// TwinCAT 3 PLC project Untitled1
// ProgramVersion: 3.1.4018.58
// libraries:
//   Tc2_Standard, * (Beckhoff Automation GmbH)
//   Tc2_System, * (Beckhoff Automation GmbH)
//   Tc2_Utilities, * (Beckhoff Automation GmbH)
//   Tc3_Module, * (Beckhoff Automation GmbH)
// project tree:
//   / PlcTask.TcTTO
//   POUs/ FB_GetEndTime.TcPOU, F_GetRampUpTimeString.TcPOU, FB_GetTimeString.TcPOU, MAIN.TcPOU
// real-time tasks:
//   TASK PlcTask: cycle T#10ms, priority 20, ADS port 350

CONFIGURATION Untitled1
    RESOURCE PLC ON TwinCAT3
        TASK PlcTask(INTERVAL := T#10ms, PRIORITY := 20);
        PROGRAM MAIN WITH PlcTask : MAIN;
    END_RESOURCE
END_CONFIGURATION

// ---- POUs/MAIN.TcPOU
PROGRAM MAIN
VAR
	bBool	: BOOL;
	iInt	: INT;
	
	fbGetEndTime: FB_GetEndTime;
	
	bTestTimeCalc	: BOOL;
	strEndTimeString	: STRING(255);
	strStartTimeString	: STRING(255);
	
	bTestGetTimeString	: BOOL;
	strTimeString		: STRING(255);
	fHours				: LREAL	:= 1.26;
END_VAR

iInt	:= iInt + 1;
IF(iInt > 100) THEN
	bBool	:= NOT(bBool); 
	iInt	:= 0;
END_IF

fbGetEndTime();
IF(bTestTimeCalc)THEN
	strEndTimeString	:= fbGetEndTime.GetEndTimeString(3900);
	bTestTimeCalc	:= FALSE;
END_IF

IF(bTestGetTimeString) THEN
	strTimeString		:= fbGetEndTime.GetTimeString(fHours);
	bTestGetTimeString	:= FALSE;
END_IF

END_PROGRAM

// ---- POUs/FB_GetEndTime.TcPOU
FUNCTION_BLOCK FB_GetEndTime	
VAR_INPUT
END_VAR
VAR
	
	// Variables for get end time
	
	diMinutesToWait		: DINT;
	ftTargetTime		: T_FILETIME64;
	stTargetTime		: TIMESTRUCT;
	strTargetTimeString		: STRING(255);
	strPrettyEndTimeString	: STRING(255);
	
	strYear	: STRING;
	strMonth: STRING;
	strDay	: STRING;
	strHour	: STRING;
	strMinute: STRING;
	strSecond: STRING;
	strMiliSecond: STRING;
	
	
	taYear	: T_Arg;
	taMonth : T_Arg;
	taDay	: T_Arg;
	taHour	: T_Arg;
	taMinute: T_Arg;
	taSecond: T_Arg;
	taMiliSecond: T_Arg;
	
	iMonth	: INT;
	
	iFindPos	: INT;
	strResidual	: STRING(255);
	
	
	fbGetTime	: NT_GetTime;
	iGetTimeToggle	: UDINT;
	bTriggerGetTime	: BOOL;
	//fbFprintf	: FB_FormatString2;
	
	
	// Variable for get time string
	fFractionalTime		: LREAL;
	dwFractionalTime	: DWORD;
	tFractionalTime		: TIME;

	sFractionalTimeString	: STRING;
	
	sMinutes	: STRING(255);
	sSecond		: STRING(255);
	
	sResidual	: STRING(255);
	
	iCharIndex	: INT;

	diMinutes	: DINT;
	iSeconds	: INT;
	
	diHours		: DINT;
	fMinutes	: LREAL;

	sDescriptiveHourLabel	: STRING;
	
END_VAR

iGetTimeToggle	:= iGetTimeToggle	+ 1;
IF(iGetTimeToggle > 10000) THEN
	bTriggerGetTime	:= NOT(bTriggerGetTime);
	iGetTimeToggle	:= 0;
END_IF

// Run fbGetTime to keep an up to date time reference 
fbGetTime(START:=bTriggerGetTime);

METHOD GetEndTimeString : STRING(255)
VAR_INPUT
		fWaitSeconds: LREAL;
END_VAR
diMinutesToWait	:= LREAL_TO_DINT(fWaitSeconds / 60);
ftTargetTime := F_TranslateFileTime64Bias(in:=SYSTEMTIME_TO_FILETIME64(fbGetTime.TIMESTR),bias:=diMinutesToWait,toUTC:=TRUE);
stTargetTime := FILETIME64_TO_SYSTEMTIME(ftTargetTime);
strTargetTimeString	:= SYSTEMTIME_TO_STRING(stTargetTime);

strResidual	:= strTargetTimeString;

// Seperate the string at the year month dash
iFindPos	:= FIND(strResidual,'-');
strYear 	:= LEFT(LEFT(strResidual,iFindPos),4);
strResidual	:= RIGHT(strResidual,LEN(strResidual)-iFindPos);

// Seperate the residual string at the month day dash
iFindPos	:= FIND(strResidual,'-');
strMonth 	:= LEFT(LEFT(strResidual,iFindPos),2);
strResidual	:= RIGHT(strResidual,LEN(strResidual)-iFindPos);

iMonth	:= STRING_TO_INT(strMonth);
CASE iMonth OF 
	01:
		strMonth	:= 'January';
	02:
		strMonth	:= 'February';
	03:
		strMonth	:= 'March';
	04:
		strMonth	:= 'April';
	05:
		strMonth	:= 'May';
	06:
		strMonth	:= 'June';
	07:
		strMonth	:= 'July';
	08:
		strMonth	:= 'August';
	09:
		strMonth	:= 'September';
	10:
		strMonth	:= 'October';
	11:
		strMonth	:= 'November';
	12:
		strMonth	:= 'December';
	ELSE
		strMonth	:= INT_TO_STRING(iMonth);	
END_CASE

// Seperate the residual string at the day hour dash
iFindPos	:= FIND(strResidual,'-');
strDay 		:= LEFT(LEFT(strResidual,iFindPos),2);
strResidual	:= RIGHT(strResidual,LEN(strResidual)-iFindPos);

// Seperate the residual string at the hour minute colon
iFindPos	:= FIND(strResidual,':');
strHour 	:= LEFT(LEFT(strResidual,iFindPos),2);
strResidual	:= RIGHT(strResidual,LEN(strResidual)-iFindPos);

// Seperate the residual string at the minute second colon
iFindPos	:= FIND(strResidual,':');
strMinute 	:= LEFT(LEFT(strResidual,iFindPos),2);
strResidual	:= RIGHT(strResidual,LEN(strResidual)-iFindPos);

// Seperate the residual string at the second mili-second point
iFindPos	:= FIND(strResidual,'.');
strSecond 	:= LEFT(LEFT(strResidual,iFindPos),2);
strResidual	:= RIGHT(strResidual,LEN(strResidual)-iFindPos);

// Residual string is the Miliseconds
strMiliSecond	:= strResidual;
(*
taYear	:= F_STRING(strYear);
taMonth	:= F_STRING(strMonth);
taDay	:= F_STRING(strYear);
taHour	:= F_STRING(strHour);
taMinute:= F_STRING(strMinute);
*)
strPrettyEndTimeString := CONCAT(CONCAT(CONCAT(CONCAT(CONCAT(CONCAT(CONCAT(CONCAT(CONCAT('',strDay),' of '),strMonth),' '),strYear),' at '),strHour),' : '),strMinute);


GetEndTimeString	:= strPrettyEndTimeString;
END_METHOD

METHOD GetTimeString : STRING(255)
VAR_INPUT
	fHours	: LREAL;
END_VAR
// Calculate time in Hours
// Convert time to ms 
fFractionalTime	:= fHours * 3.6E6;

// Convert to DW 
dwFractionalTime	:= LREAL_TO_DWORD(fFractionalTime);

// Convert to time
tFractionalTime		:= DWORD_TO_TIME(dwFractionalTime);

// Convert to string 
sFractionalTimeString := TIME_TO_STRING(tFractionalTime);


// Seperate the residual string at the minute second colon
iFindPos	:= FIND(strResidual,':');
strMinute 	:= LEFT(LEFT(strResidual,iFindPos),2);
strResidual	:= RIGHT(strResidual,LEN(strResidual)-iFindPos);

// Discard the T# at the start of the string
sResidual	:= sFractionalTimeString;
iCharIndex	:= FIND(STR2:= '#',STR1:= sResidual);
sResidual	:= RIGHT(sResidual,LEN(sResidual)-iCharIndex);

// Extract the minutes string
iCharIndex	:= FIND(STR2:= 'm',STR1:= sResidual);
sMinutes 	:= LEFT(sResidual,iCharIndex-1);
sResidual	:= RIGHT(sResidual,LEN(sResidual)-iCharIndex);

// Extract the seconds string
iCharIndex	:= FIND(STR2:= 's',STR1:= sResidual);
sSecond 	:= LEFT(LEFT(sResidual,iCharIndex),2);
sResidual	:= RIGHT(sResidual,LEN(sResidual)-iCharIndex);

diMinutes	:= STRING_TO_DINT(sMinutes);
iSeconds	:= STRING_TO_INT(sSecond);

fMinutes	:= DINT_TO_LREAL(diMinutes);

// Calculate the number of hours
diHours	:= TRUNC(fMinutes / 60);

// Calculate the number of minutes 
diMinutes	:= diMinutes - (diHours * 60);

IF(diHours > 1) THEN
	sDescriptiveHourLabel	:= 'Hours';
ELSE
	sDescriptiveHourLabel	:= 'Hour';
END_IF


//strFractionalTimeString	:= LREAL_TO_STRING(fFractionalTime);

//F_GetRampUpTimeString	:= CONCAT(STR1:='Machine is Ramping Up. Load application required in  ',STR2:= CONCAT(STR1:= INT_TO_STRING(iHours), STR2:= (CONCAT(STR1:= ' Hours and ', STR2:=(CONCAT(STR1:= INT_TO_STRING(iMinutes),STR2:= ' Minutes.'))))));

GetTimeString	:= CONCAT(CONCAT('',CONCAT(CONCAT(DINT_TO_STRING(diHours),CONCAT(CONCAT(' ',sDescriptiveHourLabel),' and  ')),DINT_TO_STRING(diMinutes))),' Minutes');
END_METHOD

END_FUNCTION_BLOCK

// ---- POUs/F_GetRampUpTimeString.TcPOU
FUNCTION F_GetRampUpTimeString : STRING
VAR_INPUT
	fTargetTemp	: LREAL;
	fRampRate	: LREAL; 
	fCurrentTemp: LREAL;
END_VAR
VAR
	fFractionalTime		: LREAL;
	dwFractionalTime	: DWORD;
	tFractionalTime		: TIME;
	sFractionalTime		: STRING;
	
	mCharIndex	: INT;
	iHours		: INT;
	iMinutes	: INT;
	strFractionalTimeString	: STRING;
	strTrimmedTimeString	: STRING;
END_VAR

(*
// Calculate time in Hours
IF(stPlatform.stTestController.stOutputs.eTestState = E_TestStates.eTS_RampUp) THEN
	fFractionalTime := ((fTargetTemp - fCurrentTemp) / fRampRate) + stPlatform.stTestController.stInputs.fSoakTime;
ELSE
	fFractionalTime := stPlatform.stTestController.stInputs.fSoakTime - (stPlatform.stTestController.stInternal.fSoakTimer / 3600);
END_IF
// Convert time to ms 
fFractionalTime	:= fFractionalTime * 3.6E6;

// Convert to DW 
dwFractionalTime	:= LREAL_TO_DWORD(fFractionalTime);

// Convert to time
tFractionalTime		:= DWORD_TO_TIME(dwFractionalTime);

// Convert to string 
strFractionalTimeString := TIME_TO_STRING(tFractionalTime);

mCharIndex	:= FIND(STR2:= 'm',STR1:= strFractionalTimeString);
strTrimmedTimeString	:= LEFT(STR:=strFractionalTimeString,SIZE:=mCharIndex);

//strFractionalTimeString	:= LREAL_TO_STRING(fFractionalTime);

//F_GetRampUpTimeString	:= CONCAT(STR1:='Machine is Ramping Up. Load application required in  ',STR2:= CONCAT(STR1:= INT_TO_STRING(iHours), STR2:= (CONCAT(STR1:= ' Hours and ', STR2:=(CONCAT(STR1:= INT_TO_STRING(iMinutes),STR2:= ' Minutes.'))))));

F_GetRampUpTimeString	:= CONCAT(STR1:='Machine is Ramping Up. Load application required in  ',STR2:= strTrimmedTimeString);

*)

END_FUNCTION

// ---- POUs/FB_GetTimeString.TcPOU
FUNCTION FB_GetTimeString : STRING(255)
VAR_INPUT
	fHours	: LREAL;
END_VAR
VAR
	fFractionalTime		: LREAL;
	dwFractionalTime	: DWORD;
	tFractionalTime		: TIME;
	
	
	sFractionalTime		: STRING;
	
	mCharIndex		: INT;
	iSeconds		: INT;
	iMinutes		: INT;
	iMiliSeconds	: INT;
	
	strFractionalTimeString	: STRING;
	strTrimmedTimeString	: STRING;
END_VAR

// Calculate time in Hours
// Convert time to ms 
fFractionalTime	:= fHours * 3.6E6;

// Convert to DW 
dwFractionalTime	:= LREAL_TO_DWORD(fFractionalTime);

// Convert to time
tFractionalTime		:= DWORD_TO_TIME(dwFractionalTime);

// Convert to string 
strFractionalTimeString := TIME_TO_STRING(tFractionalTime);

mCharIndex	:= FIND(STR2:= 'm',STR1:= strFractionalTimeString);
strTrimmedTimeString	:= LEFT(STR:=strFractionalTimeString,SIZE:=mCharIndex);

//strFractionalTimeString	:= LREAL_TO_STRING(fFractionalTime);

//F_GetRampUpTimeString	:= CONCAT(STR1:='Machine is Ramping Up. Load application required in  ',STR2:= CONCAT(STR1:= INT_TO_STRING(iHours), STR2:= (CONCAT(STR1:= ' Hours and ', STR2:=(CONCAT(STR1:= INT_TO_STRING(iMinutes),STR2:= ' Minutes.'))))));

FB_GetTimeString	:= CONCAT('',strFractionalTimeString);

END_FUNCTION
